TYPE ST_PackItem :
STRUCT
	Identity				: 	ST_PackIdentity;
	ItemState				:	STRING(15);
	RejectReason			: T_FSS_RejecCode;
	TimeStamp				: T_ISO8601Time;
	NoRead				:	STRING(5);

END_STRUCT
END_TYPE

(* stored: Version 1.1.0.1
   DUT ST_PackItem: Id {aa6910d5-bc6b-4600-8ce6-506094b95d93} *)
